FUNCTION F_OR_REF : BOOL
VAR_IN_OUT
	bValueRoot		: BOOL;
END_VAR
VAR_INPUT
	bValueCombine	: BOOL;
END_VAR

bValueRoot := bValueRoot OR bValueCombine;

END_FUNCTION

(* stored: Version 1.1.0.1, ProductVersion 3.1.4024.11
   POU F_OR_REF: Id {ba14dfb6-1b0e-4f51-b8b3-3eb9f786bd57}, SpecialFunc None *)
